// TIA Portal V17 export
// export: Created 2021-12-03T08:08:02.54171Z, ExportSetting WithDefaults, DisplayName Totally Integrated Automation Portal, DisplayVersion V17, DisplayName TIA Portal Openness, DisplayVersion V17, DisplayName TIA Portal Version Control Interface, DisplayVersion V17, DisplayName STEP 7 Professional, DisplayVersion V17, DisplayName STEP 7 Safety, DisplayVersion V17, DisplayName WinCC Advanced, DisplayVersion V17
VAR_GLOBAL   // PLC tag table "FailSafe_DO"
   O_Power_AccConsol AT %Q50.3 : Bool;   // 230 VAC Power Accelerator Console NA2-2Q3
   O_PowerChiller AT %Q50.1 : Bool;   // 400 VAC Power Chiller NA2-1Q5
   O_PowerConveyor AT %Q50.2 : Bool;   // 400 VAC Power Conveyor NA2-1Q7
   O_PowerModulator AT %Q50.0 : Bool;   // 400 VAC Power Modulator NA2-1Q3
   O_PowerModulator1P AT %Q50.5 : Bool;   // 230 VAC Power Modulator
   O_PowerXRayUnit AT %Q50.4 : Bool;   // 230 VAC Power X-Ray Unit NA2-2Q7
   O_ChilVlv_PwrOn AT %Q50.6 : Bool;   // 230 VAC Power Chiller Valve
   O_ModSwic_PwrOn AT %Q50.7 : Bool;   // 230 VAC Power Modulator Switch
   O_AccIntrlck AT %Q51.0 : Bool;   // Interlock Accelerator
   O_SpareIntrlck AT %Q51.1 : Bool;   // Interlock Spare
END_VAR
